{attribute addProperty BoxType "EL2262-0000-0004"}
{attribute addProperty Id "StartTimeNextOutputAT %I*UDINT324"}
{attribute addProperty CRC "3268638497"}
{attribute addProperty SizeInBites "32"}
{attribute addProperty SizeInBytes "4"}
TYPE StartTimeNextOutput_C2D37721 :
STRUCT
	{attribute addProperty Name "StartTimeNextOutput"}
	StartTimeNextOutput AT %I* : UDINT;
END_STRUCT
END_TYPE

(* stored: Version 1.2.0.0, ProductVersion 3.1.4024.9
   DUT StartTimeNextOutput_C2D37721: Id {2415771d-779c-4418-8aa6-c6f2c1174734} *)
